TYPE ST_Issue94_Byte :
STRUCT
	ByteValue : byte;
END_STRUCT
END_TYPE

(* stored: Version 1.1.0.1, ProductVersion 3.1.4024.9
   DUT ST_Issue94_Byte: Id {e12f220e-f2ce-4daa-8a73-4e3071cb785e} *)
